// TwinCAT 3 PLC project TimeProjectPlc
// ProgramVersion: 3.1.4024.0
// libraries:
//   Tc2_Standard, * (Beckhoff Automation GmbH)
//   Tc2_System, * (Beckhoff Automation GmbH)
//   Tc2_Utilities, * (Beckhoff Automation GmbH)
//   Tc3_Module, * (Beckhoff Automation GmbH)
// project tree:
//   DUTs/ E_EventType.TcDUT, ST_Event.TcDUT
//   / PlcTask.TcTTO
//   POUs/ FB_EventLogger.TcPOU, FB_CsvPersistentEventStorage.TcPOU, F_GetSystemDateAndTime.TcPOU, I_PersistentEventStorage.TcIO, MAIN.TcPOU
// real-time tasks:
//   TASK PlcTask: cycle T#10ms, priority 20, ADS port 350

CONFIGURATION TimeProjectPlc
    RESOURCE PLC ON TwinCAT3
        TASK PlcTask(INTERVAL := T#10ms, PRIORITY := 20);
        PROGRAM MAIN WITH PlcTask : MAIN;
    END_RESOURCE
END_CONFIGURATION

// ---- DUTs/E_EventType.TcDUT
{attribute 'qualified_only'}
{attribute 'strict'}
{attribute 'to_string'}
TYPE E_EventType :
(
	Alarm := 0,
	Message := 1
);
END_TYPE

// ---- DUTs/ST_Event.TcDUT
TYPE ST_Event :
STRUCT
	eEventType : E_EventType;
	eEventSeverity : TcEventSeverity;
	nEventIdentity : UDINT;
	sEventText : STRING(255);
	dtTimestamp : DATE_AND_TIME;
END_STRUCT
END_TYPE

// ---- POUs/I_PersistentEventStorage.TcIO
INTERFACE I_PersistentEventStorage

METHOD StoreEvent
VAR_INPUT
	stEvent : ST_Event;
END_VAR
END_METHOD

END_INTERFACE

// ---- POUs/MAIN.TcPOU
PROGRAM MAIN
VAR
	bAddEvent : BOOL;
	rtrigAddEvent : R_TRIG;
	
	eEventType : E_EventType := E_EventType.Alarm;
	eEventSeverity : TcEventSeverity := TcEventSeverity.Error;
	nEventIdentity : UDINT := 42;;
	sEventText : STRING(255) := 'This is a scary event.';
	
	fbXmlPersistentEventStorage : FB_CsvPersistentEventStorage;
	fbEventLogger : FB_EventLogger(fbXmlPersistentEventStorage);
END_VAR


rtrigAddEvent(CLK := bAddEvent);

IF rtrigAddEvent.Q THEN
	fbEventLogger.AddEvent(
		eEventType:= eEventType,
		eEventSeverity:= eEventSeverity,
		nEventIdentity:= nEventIdentity,
		sEventText:= sEventText);
END_IF

END_PROGRAM

// ---- POUs/FB_CsvPersistentEventStorage.TcPOU
FUNCTION_BLOCK FB_CsvPersistentEventStorage IMPLEMENTS I_PersistentEventStorage
VAR_INPUT
END_VAR
VAR_OUTPUT
END_VAR
VAR
END_VAR

{warning 'add method implementation '}
METHOD StoreEvent
VAR_INPUT
	stEvent	: ST_Event;
END_VAR
END_METHOD

END_FUNCTION_BLOCK

// ---- POUs/FB_EventLogger.TcPOU
FUNCTION_BLOCK FB_EventLogger
VAR
	aEventBuffer : ARRAY[1..MAXIMUM_SIZE_OF_EVENT_BUFFER] OF ST_Event;
	nCurrentEventBufferIndex : INT := 0; 
	_PersistentEventStorage : I_PersistentEventStorage;
END_VAR
VAR CONSTANT
	MAXIMUM_SIZE_OF_EVENT_BUFFER : INT := 100;
END_VAR

(* Returns TRUE if add was successful and FALSE if buffer is full *)
METHOD PUBLIC AddEvent : BOOL
VAR_INPUT
	eEventType : E_EventType;
	eEventSeverity : TcEventSeverity;
	nEventIdentity : UDINT;
	sEventText : STRING(255);
END_VAR
VAR
	stNewEvent : REFERENCE TO ST_Event;
END_VAR
AddEvent := FALSE;

IF IsEventBufferFull() THEN
	RETURN;
END_IF

// Allocate space for a new event in the event buffer
nCurrentEventBufferIndex := nCurrentEventBufferIndex + 1;
stNewEvent REF= aEventBuffer[nCurrentEventBufferIndex];

stNewEvent.eEventType := eEventType;
stNewEvent.eEventSeverity := eEventSeverity;
stNewEvent.nEventIdentity := nEventIdentity;
stNewEvent.sEventText := sEventText;
stNewEvent.dtTimestamp := F_GetSystemDateAndTime();

_PersistentEventStorage.StoreEvent(stEvent := stNewEvent);

AddEvent := TRUE;
END_METHOD

METHOD FB_init : BOOL
VAR_INPUT
	bInitRetains : BOOL; // if TRUE, the retain variables are initialized (warm start / cold start)
	bInCopyCode : BOOL;  // if TRUE, the instance afterwards gets moved into the copy code (online change)
	iPersistentEventStorage : I_PersistentEventStorage;
END_VAR
_PersistentEventStorage := iPersistentEventStorage;
END_METHOD

METHOD PUBLIC IsEventBufferFull : BOOL
IsEventBufferFull := (nCurrentEventBufferIndex + 1) > MAXIMUM_SIZE_OF_EVENT_BUFFER;
END_METHOD

END_FUNCTION_BLOCK

// ---- POUs/F_GetSystemDateAndTime.TcPOU
FUNCTION F_GetSystemDateAndTime : DATE_AND_TIME
VAR
	fbGETSYSTEMTIME : GETSYSTEMTIME;
	stFileTime : T_FILETIME;
END_VAR

fbGETSYSTEMTIME(timeLoDW => stFileTime.dwLowDateTime,
				timeHiDW => stFileTime.dwHighDateTime);

F_GetSystemDateAndTime := FILETIME_TO_DT(fileTime := stFileTime);

END_FUNCTION
